// TIA Portal V16 export
// export: Created 2022-09-01T13:36:57.6832982Z, ExportSetting WithDefaults, DisplayName Totally Integrated Automation Portal, DisplayVersion V16, DisplayName TIA Portal Version Control Interface, DisplayVersion V16, DisplayName TIA Portal Openness, DisplayVersion V16, DisplayName STEP 7 Professional, DisplayVersion V16, DisplayName STEP 7 Safety, DisplayVersion V16, DisplayName WinCC Advanced, DisplayVersion V16
FUNCTION "Estab_Níveis" : Void   // FC20, LAD
TITLE = Protege equipamentos e evita transbordo em modo manual
{ S7_Optimized_Access := 'TRUE' }
VERSION : 0.1
// stored: AutoNumber true, IsIECCheckEnabled false, SetENOAutomatically false, UDAEnableTagReadback false
BEGIN

REGION Network 1: LSL001
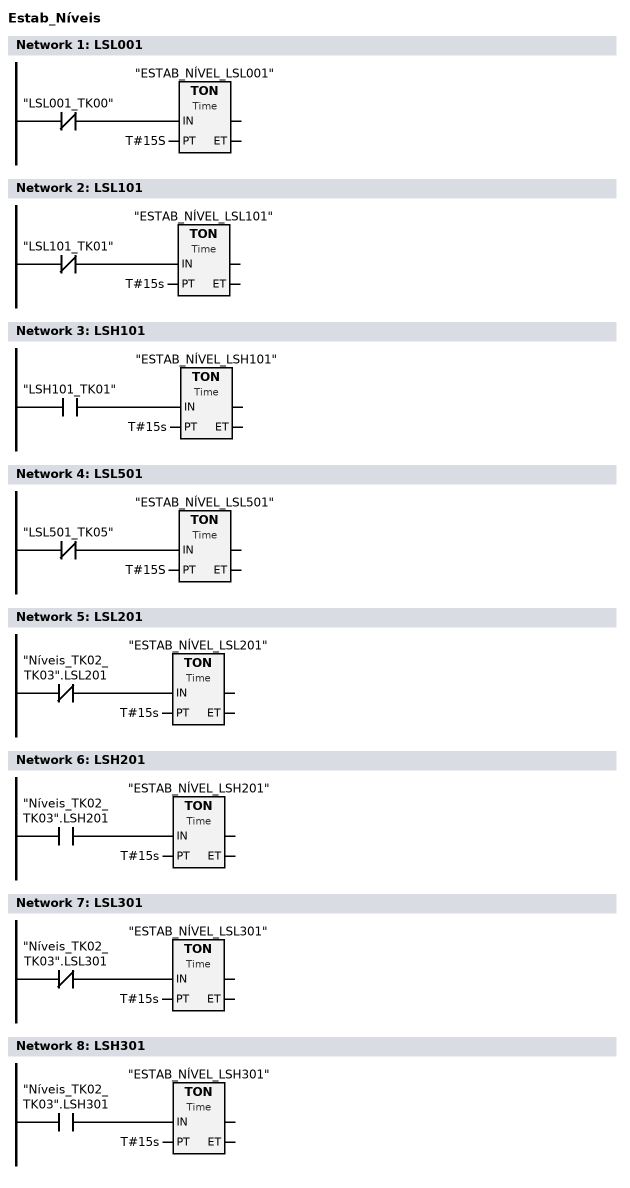
   RUNG wire#powerrail
      I_Contact( "LSL001_TK00" )
      { S7_Templates := "time_type := Time" } "ESTAB_NÍVEL_LSL001".TON(pt := T#15S, et =>)
   END_RUNG
   // the same network as SCL:
   "ESTAB_NÍVEL_LSL001".TON(IN := NOT "LSL001_TK00", PT := T#15S);
END_REGION

REGION Network 2: LSL101
   RUNG wire#powerrail
      I_Contact( "LSL101_TK01" )
      { S7_Templates := "time_type := Time" } "ESTAB_NÍVEL_LSL101".TON(pt := T#15s, et =>)
   END_RUNG
   // the same network as SCL:
   "ESTAB_NÍVEL_LSL101".TON(IN := NOT "LSL101_TK01", PT := T#15s);
END_REGION

REGION Network 3: LSH101
   RUNG wire#powerrail
      Contact( "LSH101_TK01" )
      { S7_Templates := "time_type := Time" } "ESTAB_NÍVEL_LSH101".TON(pt := T#15s, et =>)
   END_RUNG
   // the same network as SCL:
   "ESTAB_NÍVEL_LSH101".TON(IN := "LSH101_TK01", PT := T#15s);
END_REGION

REGION Network 4: LSL501
   RUNG wire#powerrail
      I_Contact( "LSL501_TK05" )
      { S7_Templates := "time_type := Time" } "ESTAB_NÍVEL_LSL501".TON(pt := T#15S, et =>)
   END_RUNG
   // the same network as SCL:
   "ESTAB_NÍVEL_LSL501".TON(IN := NOT "LSL501_TK05", PT := T#15S);
END_REGION

REGION Network 5: LSL201
   RUNG wire#powerrail
      I_Contact( "Níveis_TK02_TK03".LSL201 )
      { S7_Templates := "time_type := Time" } "ESTAB_NÍVEL_LSL201".TON(pt := T#15s, et =>)
   END_RUNG
   // the same network as SCL:
   "ESTAB_NÍVEL_LSL201".TON(IN := NOT "Níveis_TK02_TK03".LSL201, PT := T#15s);
END_REGION

REGION Network 6: LSH201
   RUNG wire#powerrail
      Contact( "Níveis_TK02_TK03".LSH201 )
      { S7_Templates := "time_type := Time" } "ESTAB_NÍVEL_LSH201".TON(pt := T#15s, et =>)
   END_RUNG
   // the same network as SCL:
   "ESTAB_NÍVEL_LSH201".TON(IN := "Níveis_TK02_TK03".LSH201, PT := T#15s);
END_REGION

REGION Network 7: LSL301
   RUNG wire#powerrail
      I_Contact( "Níveis_TK02_TK03".LSL301 )
      { S7_Templates := "time_type := Time" } "ESTAB_NÍVEL_LSL301".TON(pt := T#15s, et =>)
   END_RUNG
   // the same network as SCL:
   "ESTAB_NÍVEL_LSL301".TON(IN := NOT "Níveis_TK02_TK03".LSL301, PT := T#15s);
END_REGION

REGION Network 8: LSH301
   RUNG wire#powerrail
      Contact( "Níveis_TK02_TK03".LSH301 )
      { S7_Templates := "time_type := Time" } "ESTAB_NÍVEL_LSH301".TON(pt := T#15s, et =>)
   END_RUNG
   // the same network as SCL:
   "ESTAB_NÍVEL_LSH301".TON(IN := "Níveis_TK02_TK03".LSH301, PT := T#15s);
END_REGION
END_FUNCTION
